FUNCTION_BLOCK PUBLIC FB_Lamp
VAR_OUTPUT
	byLevel			: BYTE;
END_VAR

PROPERTY PUBLIC Level : BYTE
GET
Level := byLevel;
END_GET
END_PROPERTY

METHOD PUBLIC SetLevel : BOOL
VAR_INPUT
	byNewLevel			: BYTE;
END_VAR
byLevel := byNewLevel;
END_METHOD

END_FUNCTION_BLOCK

(* stored: Version 1.1.0.1, ProductVersion 3.1.4020.3
   POU FB_Lamp: Id {c9363aa1-33e3-41da-adea-7faeb59d6855}, SpecialFunc None
   Property Level: Id {14dcd475-0945-4468-8762-cbfbbeb1403d}
   Get Get: Id {48f1de5c-993e-42ec-a2e6-7dc3b36570be}
   Method SetLevel: Id {97c2b33b-5c80-46f7-8f00-32f4f1bdd6a5} *)
